TYPE ST_Filter_Current_Hexapod_Robot_Input :
STRUCT
	Current_Motor: matrix_18_real_T;
END_STRUCT
END_TYPE

(* stored: Version 1.1.0.1, ProductVersion 3.1.4020.12
   DUT ST_Filter_Current_Hexapod_Robot_Input: Id {43428ddf-1a61-4b6d-ab5c-19d637c6725e} *)
